// TIA Portal V18 program export: 0 tag tables, 0 data types, 0 data blocks, 3 code blocks (in call order from the OBs), 2 instance data blocks

ORGANIZATION_BLOCK "Main"   // OB1, LAD, ProgramCycle
TITLE = "Main Program Sweep (Cycle)"
{ S7_Optimized_Access := 'TRUE' }
// stored: SetENOAutomatically false
   VAR_INPUT
      Initial_Call : Bool;   // Initial call of this OB
      Remanence : Bool;   // =True, if remanent data are available
   END_VAR
BEGIN

REGION Network 1
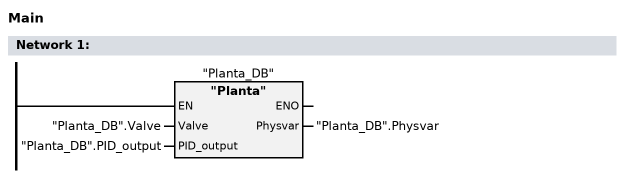
   RUNG wire#powerrail
      "Planta_DB"(Valve := "Planta_DB".Valve, PID_output := "Planta_DB".PID_output, Physvar => "Planta_DB".Physvar)
   END_RUNG
   // the same network as SCL:
   "Planta_DB"(Valve := "Planta_DB".Valve, PID_output := "Planta_DB".PID_output, Physvar => "Planta_DB".Physvar);   // "Planta"
END_REGION
END_ORGANIZATION_BLOCK

FUNCTION_BLOCK "Planta"   // FB2, LAD
{ S7_Optimized_Access := 'FALSE' }
// stored: SetENOAutomatically false
   VAR_INPUT
      Valve : Bool;
      PID_output : Real;
   END_VAR
   VAR_OUTPUT
      Physvar : Real;
   END_VAR
   VAR
      F1 : Bool;
      F2 : Bool;
      F3 : Bool;
      F4 : Bool;
      F5 : Bool;
      F6 : Bool;
      LL : Real := 20.0;
      L : Real := 40.0;
      H : Real := 60.0;
      HH : Real := 80.0;
      LL_M : Real := 0.01;
      L_M : Real := 0.05;
      H_M : Real := 0.1;
      HH_M : Real := 0.2;
      MAX_M : Real := 0.5;
      Out_M : Real := 0.1;
   END_VAR
   VAR_TEMP   // added for the SCL form of the ladder/FBD networks
      _w1 : Bool;
   END_VAR
BEGIN

REGION Network 1
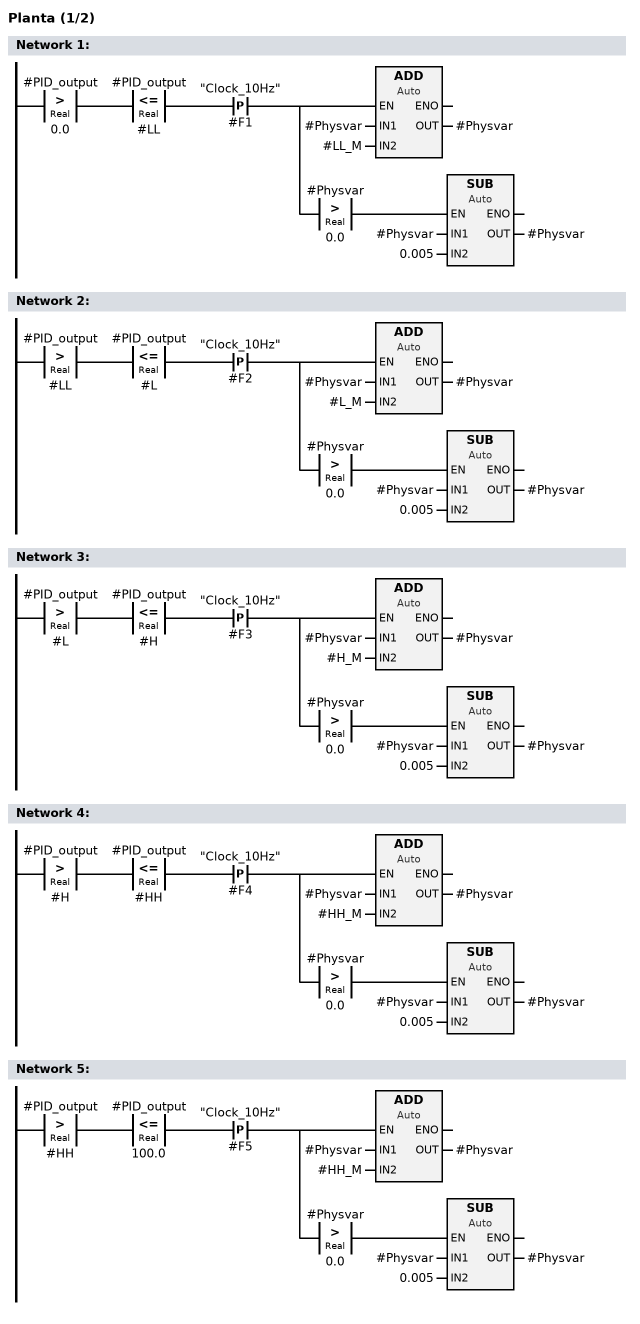
   RUNG wire#powerrail
      { S7_Templates := "SrcType := Real" } GT_Contact(in1 := #PID_output, in2 := 0.0)
      { S7_Templates := "SrcType := Real" } LE_Contact(in1 := #PID_output, in2 := #LL)
      P_Contact(operand := "Clock_10Hz", bit := #F1)
      wire#w1
      Add(in1 := #Physvar, in2 := #LL_M, out => #Physvar)
   END_RUNG
   RUNG wire#w1
      { S7_Templates := "SrcType := Real" } GT_Contact(in1 := #Physvar, in2 := 0.0)
      Sub(in1 := #Physvar, in2 := 0.005, out => #Physvar)
   END_RUNG
   // the same network as SCL:
   #_w1 := (#PID_output > 0.0) AND (#PID_output <= #LL) AND "Clock_10Hz" AND NOT #F1;   // rising edge of "Clock_10Hz"
   #F1 := "Clock_10Hz";
   IF #_w1 THEN #Physvar := #Physvar + #LL_M; END_IF;
   IF #_w1 AND (#Physvar > 0.0) THEN #Physvar := #Physvar - 0.005; END_IF;
END_REGION

REGION Network 2
   RUNG wire#powerrail
      { S7_Templates := "SrcType := Real" } GT_Contact(in1 := #PID_output, in2 := #LL)
      { S7_Templates := "SrcType := Real" } LE_Contact(in1 := #PID_output, in2 := #L)
      P_Contact(operand := "Clock_10Hz", bit := #F2)
      wire#w1
      Add(in1 := #Physvar, in2 := #L_M, out => #Physvar)
   END_RUNG
   RUNG wire#w1
      { S7_Templates := "SrcType := Real" } GT_Contact(in1 := #Physvar, in2 := 0.0)
      Sub(in1 := #Physvar, in2 := 0.005, out => #Physvar)
   END_RUNG
   // the same network as SCL:
   #_w1 := (#PID_output > #LL) AND (#PID_output <= #L) AND "Clock_10Hz" AND NOT #F2;   // rising edge of "Clock_10Hz"
   #F2 := "Clock_10Hz";
   IF #_w1 THEN #Physvar := #Physvar + #L_M; END_IF;
   IF #_w1 AND (#Physvar > 0.0) THEN #Physvar := #Physvar - 0.005; END_IF;
END_REGION

REGION Network 3
   RUNG wire#powerrail
      { S7_Templates := "SrcType := Real" } GT_Contact(in1 := #PID_output, in2 := #L)
      { S7_Templates := "SrcType := Real" } LE_Contact(in1 := #PID_output, in2 := #H)
      P_Contact(operand := "Clock_10Hz", bit := #F3)
      wire#w1
      Add(in1 := #Physvar, in2 := #H_M, out => #Physvar)
   END_RUNG
   RUNG wire#w1
      { S7_Templates := "SrcType := Real" } GT_Contact(in1 := #Physvar, in2 := 0.0)
      Sub(in1 := #Physvar, in2 := 0.005, out => #Physvar)
   END_RUNG
   // the same network as SCL:
   #_w1 := (#PID_output > #L) AND (#PID_output <= #H) AND "Clock_10Hz" AND NOT #F3;   // rising edge of "Clock_10Hz"
   #F3 := "Clock_10Hz";
   IF #_w1 THEN #Physvar := #Physvar + #H_M; END_IF;
   IF #_w1 AND (#Physvar > 0.0) THEN #Physvar := #Physvar - 0.005; END_IF;
END_REGION

REGION Network 4
   RUNG wire#powerrail
      { S7_Templates := "SrcType := Real" } GT_Contact(in1 := #PID_output, in2 := #H)
      { S7_Templates := "SrcType := Real" } LE_Contact(in1 := #PID_output, in2 := #HH)
      P_Contact(operand := "Clock_10Hz", bit := #F4)
      wire#w1
      Add(in1 := #Physvar, in2 := #HH_M, out => #Physvar)
   END_RUNG
   RUNG wire#w1
      { S7_Templates := "SrcType := Real" } GT_Contact(in1 := #Physvar, in2 := 0.0)
      Sub(in1 := #Physvar, in2 := 0.005, out => #Physvar)
   END_RUNG
   // the same network as SCL:
   #_w1 := (#PID_output > #H) AND (#PID_output <= #HH) AND "Clock_10Hz" AND NOT #F4;   // rising edge of "Clock_10Hz"
   #F4 := "Clock_10Hz";
   IF #_w1 THEN #Physvar := #Physvar + #HH_M; END_IF;
   IF #_w1 AND (#Physvar > 0.0) THEN #Physvar := #Physvar - 0.005; END_IF;
END_REGION

REGION Network 5
   RUNG wire#powerrail
      { S7_Templates := "SrcType := Real" } GT_Contact(in1 := #PID_output, in2 := #HH)
      { S7_Templates := "SrcType := Real" } LE_Contact(in1 := #PID_output, in2 := 100.0)
      P_Contact(operand := "Clock_10Hz", bit := #F5)
      wire#w1
      Add(in1 := #Physvar, in2 := #HH_M, out => #Physvar)
   END_RUNG
   RUNG wire#w1
      { S7_Templates := "SrcType := Real" } GT_Contact(in1 := #Physvar, in2 := 0.0)
      Sub(in1 := #Physvar, in2 := 0.005, out => #Physvar)
   END_RUNG
   // the same network as SCL:
   #_w1 := (#PID_output > #HH) AND (#PID_output <= 100.0) AND "Clock_10Hz" AND NOT #F5;   // rising edge of "Clock_10Hz"
   #F5 := "Clock_10Hz";
   IF #_w1 THEN #Physvar := #Physvar + #HH_M; END_IF;
   IF #_w1 AND (#Physvar > 0.0) THEN #Physvar := #Physvar - 0.005; END_IF;
END_REGION

REGION Network 6
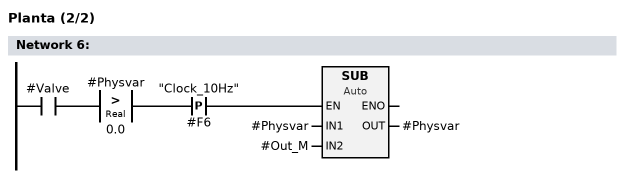
   RUNG wire#powerrail
      Contact( #Valve )
      { S7_Templates := "SrcType := Real" } GT_Contact(in1 := #Physvar, in2 := 0.0)
      P_Contact(operand := "Clock_10Hz", bit := #F6)
      Sub(in1 := #Physvar, in2 := #Out_M, out => #Physvar)
   END_RUNG
   // the same network as SCL:
   #_w1 := #Valve AND (#Physvar > 0.0) AND "Clock_10Hz" AND NOT #F6;   // rising edge of "Clock_10Hz"
   #F6 := "Clock_10Hz";
   IF #_w1 THEN #Physvar := #Physvar - #Out_M; END_IF;
END_REGION
END_FUNCTION_BLOCK

ORGANIZATION_BLOCK "Cyclic interrupt"   // OB30, LAD, CyclicInterrupt
{ S7_Optimized_Access := 'TRUE' }
// stored: SetENOAutomatically false
   VAR_INPUT
      Initial_Call : Bool;   // Initial call of this OB
      Event_Count : Int;   // Events discarded
   END_VAR
BEGIN

REGION Network 1
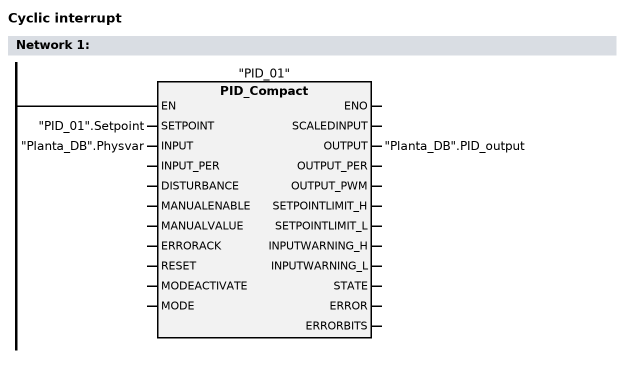
   RUNG wire#powerrail
      "PID_01".PID_Compact(Setpoint := "PID_01".Setpoint, Input := "Planta_DB".Physvar, Input_PER :=, Disturbance :=, ManualEnable :=, ManualValue :=, ErrorAck :=, Reset :=, ModeActivate :=, Mode :=, ScaledInput =>, Output => "Planta_DB".PID_output, Output_PER =>, Output_PWM =>, SetpointLimit_H =>, SetpointLimit_L =>, InputWarning_H =>, InputWarning_L =>, State =>, Error =>, ErrorBits =>)
   END_RUNG
   // the same network as SCL:
   "PID_01"(Setpoint := "PID_01".Setpoint, Input := "Planta_DB".Physvar, Output => "Planta_DB".PID_output);   // PID_Compact
END_REGION
END_ORGANIZATION_BLOCK

DATA_BLOCK "Planta_DB"   // DB2
// stored: InstanceOfName Planta, InstanceOfType FB
"Planta"
BEGIN
END_DATA_BLOCK

DATA_BLOCK "PID_01"   // DB1
// stored: InstanceOfName PID_Compact, OfSystemLibElement PID_Compact, OfSystemLibVersion 2.4
PID_Compact   // technology object, version 2.4
   // VAR_INPUT
   //    Setpoint : Real;
   //    Input : Real;
   //    Input_PER : Int;
   //    Disturbance : Real;
   //    ManualEnable : Bool;
   //    ManualValue : Real;
   //    ErrorAck : Bool;
   //    Reset : Bool;
   //    ModeActivate : Bool;
   // END_VAR
   // VAR_OUTPUT
   //    ScaledInput { ExternalWritable := 'False'} : Real;
   //    Output { ExternalWritable := 'False'} : Real;
   //    Output_PER { ExternalWritable := 'False'} : Int;
   //    Output_PWM { ExternalWritable := 'False'} : Bool;
   //    SetpointLimit_H { ExternalWritable := 'False'} : Bool;
   //    SetpointLimit_L { ExternalWritable := 'False'} : Bool;
   //    InputWarning_H { ExternalWritable := 'False'} : Bool;
   //    InputWarning_L { ExternalWritable := 'False'} : Bool;
   //    State { ExternalWritable := 'False'} : Int;
   //    Error { ExternalWritable := 'False'} : Bool;
   //    ErrorBits { ExternalWritable := 'False'} : DWord;
   // END_VAR
   // VAR_IN_OUT
   //    Mode : Int := 3;
   // END_VAR
   // VAR
   //    InternalDiagnostic : DWord;
   //    InternalVersion { ExternalWritable := 'False'} : DWord;
   //    InternalRTVersion : DWord;
   //    IntegralResetMode { S7_SetPoint := 'True'} : Int;
   //    OverwriteInitialOutputValue : Real;
   //    RunModeByStartup { S7_SetPoint := 'True'} : Bool;
   //    LoadBackUp : Bool;
   //    SetSubstituteOutput { S7_SetPoint := 'True'} : Bool;
   //    PhysicalUnit { ExternalWritable := 'False'; S7_SetPoint := 'True'} : Int;
   //    PhysicalQuantity { ExternalWritable := 'False'; S7_SetPoint := 'True'} : Int;
   //    ActivateRecoverMode { S7_SetPoint := 'True'} : Bool;
   // END_VAR
   // VAR RETAIN
   //    Warning { ExternalWritable := 'False'} : DWord;
   //    WarningInternal { ExternalWritable := 'False'} : DWord;
   // END_VAR
   // VAR
   //    Progress { ExternalWritable := 'False'} : Real;
   //    CurrentSetpoint { ExternalWritable := 'False'} : Real;
   //    CancelTuningLevel { S7_SetPoint := 'True'} : Real;
   //    SubstituteOutput { S7_SetPoint := 'True'} : Real;
   //    Config { S7_SetPoint := 'True'} : PID_CompactConfig;
   //    CycleTime { S7_SetPoint := 'True'} : PID_CycleTime;
   //    CtrlParamsBackUp { S7_SetPoint := 'True'} : PID_CompactControlParams;
   //    PIDSelfTune { S7_SetPoint := 'True'} : PID_CompactSelfTune;
   //    PIDCtrl { S7_SetPoint := 'True'} : PID_CompactControl;
   // END_VAR
   // VAR RETAIN
   //    Retain { S7_SetPoint := 'True'} : PID_CompactRetain;
   // END_VAR
BEGIN
   Config.InputPerOn := FALSE;
   Retain.CtrlParams.Gain := 39.53336;
   Retain.CtrlParams.Ti := 1.064005;
   Retain.CtrlParams.Td := 0.2380012;
   Retain.CtrlParams.TdFiltRatio := 0.1;
   Retain.CtrlParams.PWeighting := 0.58;
   Retain.CtrlParams.DWeighting := 0.0;
   Retain.CtrlParams.Cycle := 0.1000005;
END_DATA_BLOCK
